Staubli VAL3: onEnterEvent.pgx

program onEnterEvent()
  local num l_nPoint
  local bool l_bInside
  local bool l_bOk
begin
  //
  // NB sEvent is the selected
  // element in the LIST
  //
  if !cycleStatus:bSimulation
    call use:stringToArray(sTrajName+","+toString("",nPoint),sMessage)
    // reload the traj
    //call loadEditTraj(sTrajName)
    //
    call loadPage("Disk://trajectory/page_editTraj",sMessage)
    // reload the traj
    call loadEditTraj(sTrajName)
    //
    // ELEBORATE THE GIVE BACK
    //
    l_bOk=true
    toNum(sMessage[1],l_nPoint,l_bOk)
    call isAtPoint(l_nPoint,l_bInside)
    if l_bInside
      nPoint=l_nPoint
    endIf
    cls()
    use:bUseRefresh=true
    // reset the show status
    bShowStatus=false
  endIf
end
